FUNCTION_BLOCK FB_Bel_Stellwertscheck
VAR_IN_OUT
	Stellwert	: ST_Bel_Stellwert;
END_VAR

VAR_INPUT
(*	Steuerung	: ST_BHKW_Steuerung; *)
(*	Zustand	: ST_PU_Zustand; *)
	Parameter	: ST_Bel_Parameter;
END_VAR
VAR_OUTPUT
END_VAR
VAR
	Timer1			: TON;
END_VAR

Timer1(	IN := Stellwert.Betrieb = FALSE,
		PT := T#15S,
		Q => Stellwert.Freigabe_Stellwert
);

END_FUNCTION_BLOCK

(* stored: Version 1.1.0.1, ProductVersion 3.1.4024.9
   POU FB_Bel_Stellwertscheck: Id {8f265280-aa74-4a22-8dc8-9aca0f4a9bea}, SpecialFunc None *)
